FUNCTION_BLOCK L3_ReleasedMHDLR (* Basic Function Block Type *)
  (* Standard: 61499-2 *)
  (* Version 0.0, 2014-10-06, EQUEROL, UJI *)
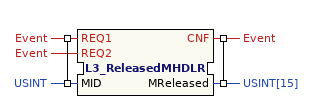
  EVENT_INPUT
    REQ1 WITH MID; (* Response from PP, released machine *)
    REQ2; (* Normal Execution Request *)
  END_EVENT
  EVENT_OUTPUT
    CNF WITH MReleased; (* Execution Confirmation *)
  END_EVENT
  VAR_INPUT
    MID : USINT; (* released machine Identifier *)
  END_VAR
  VAR_OUTPUT
    MReleased : ARRAY [0..14] OF USINT; (* Vector holding released machines since last call *)
  END_VAR
  VAR
    ReleasedMachines : ARRAY [0..14] OF USINT := [0,0,0,0,0,0,0,0,0,0,0,0,0,0,0]; (* vector holding released machines since last call *)
    i : USINT; (* loop variable *)
  END_VAR
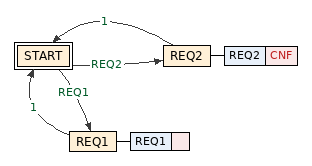
  EC_STATES
    START; (* Initial State *)
    REQ2 : REQ2 -> CNF; (* Normal execution *)
    REQ1 : REQ1;
  END_STATES
  EC_TRANSITIONS
    START TO REQ2 := REQ2;
    REQ2 TO START := 1;
    START TO REQ1 := REQ1;
    REQ1 TO START := 1;
  END_TRANSITIONS
  ALGORITHM REQ2 IN ST: (* Normally executed algorithm *)
(*This algo send to the core the released machines and resets the internal vector*)
FOR i := 0 TO 14 DO
		MReleased[i] := ReleasedMachines[i];
		ReleasedMachines[i] := 0;
END_FOR;
  END_ALGORITHM
  ALGORITHM REQ1 IN ST: (* Update released machines vector *)
IF MID>=0 AND MID <15 THEN
	ReleasedMachines[MID] := 2;
END_IF;
  END_ALGORITHM
END_FUNCTION_BLOCK
